// TwinCAT 3 PLC project Untitled1
// ProgramVersion: 3.1.4023.0
// libraries:
//   Tc2_BABasic, * (Beckhoff Automation GmbH)
//   Tc2_ControllerToolbox, * (Beckhoff Automation GmbH)
//   Tc2_MC2, * (Beckhoff Automation GmbH)
//   Tc2_NC, * (Beckhoff Automation GmbH)
//   Tc2_NCI, * (Beckhoff Automation GmbH)
//   Tc2_Standard, * (Beckhoff Automation GmbH)
//   Tc2_System, * (Beckhoff Automation GmbH)
//   Tc2_TempController, * (Beckhoff Automation GmbH)
//   Tc3_Module, * (Beckhoff Automation GmbH)
//   Tc3_mxAutomation, * (Beckhoff Automation GmbH)
//   Tc3_mxAutomationV3_0, * (Beckhoff Automation GmbH)
//   VisuDialogs, * (System)
//   PLC_EposCmdNick,1.0.0.0,TUT
//   VisuSymbols,3.5.10.0,System
// project tree:
//   / GlobalTextList.TcGTLO, PlcTask.TcTTO, Visualization Manager.TcVMO (not stored)
//   GVLs/ GVL_AxisCtrl.TcGVL, GVL_IO.TcGVL, GVL_NC.TcGVL, Scope_Variables.TcGVL
//   POUs/Backup/ PRG_ExtrusionSystem.TcPOU (not stored)
//   POUs/FB/ FB_EnableAxis.TcPOU, FB_EnableNetwork.TcPOU, FB_EPOSstates.TcPOU, FB_EPOS_Control.TcPOU, FB_ExtrusionSystem.TcPOU, FB_SimpleNciSequence.TcPOU, FB_TempControl.TcPOU, FB_ExtrusionSystemRev.TcPOU
//   POUs/ MAIN.TcPOU
//   POUs/Programs/ PRG_AxisControl.TcPOU, PRG_AxesEnable.TcPOU, PRG_ExtruderSys.TcPOU, PRG_ExtruderSys_Alt.TcPOU, PRG_Init.TcPOU, PRG_updateDrives.TcPOU
//   VISUs/ Visualization.TcVIS
// real-time tasks:
//   TASK PlcTask: cycle T#10ms, priority 20, ADS port 350
// motion (NC):
//   TASK NC-Task 1 SAF: cycle T#2ms, priority 4, ADS port 501
//   TASK NC-Task 1 SVB: cycle T#10ms, priority 8, ADS port 511
//   AXIS Axis Th1 (id 1)
//     General: UnitName=°
//     Dynamic: AccelerationMaximum=1500
//     Velo: SlowManual=60, FastManual=80, Maximum=200
//     OtherSettings: AllowMotionCmdToSlave=true, PulseDistancePos=2, PulseDistanceNeg=2
//     encoder EncType=16
//       EncPara: ScaleFactorNumerator=0.000457763671875, MaxCount=#x0000ffff
//         SoftEndMinControl: Enable=true, Range=-16
//         SoftEndMaxControl: Enable=true, Range=35
//     drive DrvType=5
//       Analog: VeloReferenz=220, TorqueSetpointScale=10, ScaleFactorActTorque=0.1
//       TimeComp: TaskDelayCycles=1
//     controller CtrType=1
//       CtrPara: PriorControlFactor=1
//         PosDiffControl: Enable=false
//         PID: PosKp=10
//         Observer: BandWidth=20
//   AXIS Axis Th2 (id 2)
//     General: UnitName=°
//     Velo: SlowManual=60, FastManual=100, Maximum=200
//     OtherSettings: AllowMotionCmdToSlave=true, PulseDistancePos=2, PulseDistanceNeg=2
//     encoder EncType=16
//       EncPara: ScaleFactorNumerator=0.000457763671875, MaxCount=#x0000ffff
//     drive DrvType=5
//       Analog: VeloReferenz=220, TorqueSetpointScale=10, ScaleFactorActTorque=0.1
//       TimeComp: TaskDelayCycles=1
//     controller CtrType=1
//       CtrPara: PriorControlFactor=1
//         PosDiffControl: Enable=false
//         PID: PosKp=10
//         Observer: BandWidth=20
//   AXIS Axis Extruder (id 3)
//     Dynamic: AccelerationMaximum=168, Acceleration=167
//     Velo: RefSearch=10, RefSync=15, SlowManual=10.1, FastManual=15, Maximum=20
//     OtherSettings: AllowMotionCmdToSlave=true
//     encoder EncType=1
//       EncPara: ScaleFactorNumerator=0.000310550364583
//         Inc: RefSoftSyncMask=#x0000ffff
//     drive DrvType=24
//       Analog: VeloReferenz=20, TorqueSetpointScale=10, ScaleFactorActTorque=0.1
//       TimeComp: TaskDelayCycles=1
//     controller CtrType=1
//       CtrPara: PriorControlFactor=1
//         PosDiffControl: Enable=false
//         Observer: BandWidth=20
//   AXIS Axis X (id 4)
//     OtherSettings: AllowMotionCmdToSlave=true
//     encoder EncType=1
//     drive DrvType=5
//       Analog: TorqueSetpointScale=10, ScaleFactorActTorque=0.1
//       TimeComp: TaskDelayCycles=1
//     controller CtrType=1
//       CtrPara: PriorControlFactor=1
//         Observer: BandWidth=20
//   AXIS Axis Z (id 5)
//     OtherSettings: AllowMotionCmdToSlave=true
//     encoder EncType=1
//     drive DrvType=5
//       Analog: TorqueSetpointScale=10, ScaleFactorActTorque=0.1
//       TimeComp: TaskDelayCycles=1
//     controller CtrType=1
//       CtrPara: PriorControlFactor=1
//         Observer: BandWidth=20
//   AXIS Axis Pitch (id 6)
//     OtherSettings: AllowMotionCmdToSlave=true
//     encoder EncType=1
//     drive DrvType=5
//       Analog: TorqueSetpointScale=10, ScaleFactorActTorque=0.1
//       TimeComp: TaskDelayCycles=1
//     controller CtrType=1
//       CtrPara: PriorControlFactor=1
//         Observer: BandWidth=20
//   AXIS Axis Roll (id 7)
//     OtherSettings: AllowMotionCmdToSlave=true
//     encoder EncType=1
//     drive DrvType=5
//       Analog: TorqueSetpointScale=10, ScaleFactorActTorque=0.1
//       TimeComp: TaskDelayCycles=1
//     controller CtrType=1
//       CtrPara: PriorControlFactor=1
//         Observer: BandWidth=20
// I/O:
//   DEVICE Device 2 (EtherCAT), AmsNetId 130.230.11.184.3.1
//     Term 17 (EK1100) [EK1100 EtherCAT Coupler (2A E-Bus)]
//       Term 16 (EL6751) [EL6751 CANopen Master]
//       Term 19 (EL3202) [EL3202 2Ch. Ana. Input PT100 (RTD)]
//       Term 20 (EL1004) [EL1004 4Ch. Dig. Input 24V, 3ms]
//       Term 21 (EL7041) [EL7041 1Ch. Stepper motor output stage (50V, 5A)]
//       Term 22 (EL2004) [EL2004 4Ch. Dig. Output 24V, 0.5A]
//       Term 23 (EL7332) [EL7332 2Ch. DC motor output stage (24V, 1.5A)]
//       Term 22 (EL9011) [EL9011 End Terminal]
//   DEVICE Device 1 (EL6751), AmsNetId 130.230.11.184.2.1
//     Box 2 (EPOS2)
//     Box 3 (EPOS2)
// variable links:
//   NC-Task 1 SAF/Axes/Axis Extruder <-> Device 2 (EtherCAT)/Term 17 (EK1100)/Term 21 (EL7041)
//     Drive/Inputs/In/nState1 @bit 3 <-> STM Status/Status/Error
//     Drive/Inputs/In/nState1 @bit 5 <-> STM Status/Status/Moving negative
//     Drive/Inputs/In/nState1 @bit 4 <-> STM Status/Status/Moving positive
//     Drive/Inputs/In/nState1 @bit 1 <-> STM Status/Status/Ready
//     Drive/Inputs/In/nState1 <-> STM Status/Status/Ready to enable
//     Drive/Inputs/In/nState1 @bit 6 <-> STM Status/Status/Torque reduced
//     Drive/Inputs/In/nState1 @bit 2 <-> STM Status/Status/Warning
//     Drive/Inputs/In/nState2 @bit 3 <-> STM Status/Status/Digital input 1
//     Drive/Inputs/In/nState2 @bit 4 <-> STM Status/Status/Digital input 2
//     Drive/Inputs/In/nState4 @bit 1 <-> WcState/InputToggle
//     Drive/Inputs/In/nState4 <-> WcState/WcState
//     Drive/Outputs/Out/nCtrl1 <-> STM Control/Control/Enable
//     Drive/Outputs/Out/nCtrl1 @bit 2 <-> STM Control/Control/Reduce torque
//     Drive/Outputs/Out/nCtrl1 @bit 1 <-> STM Control/Control/Reset
//     Drive/Outputs/Out/nDataOut2[0] <-> STM Velocity/Velocity
//     Enc/Inputs/In/nDataIn1[0] <-> ENC Status compact/Counter value
//     Enc/Inputs/In/nDataIn2[0] <-> ENC Status compact/Latch value
//     Enc/Inputs/In/nState1 @bit 4 <-> ENC Status compact/Status/Counter overflow
//     Enc/Inputs/In/nState1 @bit 3 <-> ENC Status compact/Status/Counter underflow
//     Enc/Inputs/In/nState1 @bit 7 <-> ENC Status compact/Status/Extrapolation stall
//     Enc/Inputs/In/nState1 <-> ENC Status compact/Status/Latch C valid
//     Enc/Inputs/In/nState1 @bit 1 <-> ENC Status compact/Status/Latch extern valid
//     Enc/Inputs/In/nState1 @bit 2 <-> ENC Status compact/Status/Set counter done
//     Enc/Inputs/In/nState2 @bit 4 <-> ENC Status compact/Status/Status of extern latch
//     Enc/Inputs/In/nState2 <-> ENC Status compact/Status/Status of input A
//     Enc/Inputs/In/nState2 @bit 1 <-> ENC Status compact/Status/Status of input B
//     Enc/Inputs/In/nState2 @bit 2 <-> ENC Status compact/Status/Status of input C
//     Enc/Inputs/In/nState4 @bit 1 <-> WcState/InputToggle
//     Enc/Inputs/In/nState4 <-> WcState/WcState
//     Enc/Outputs/Out/nCtrl1 <-> ENC Control compact/Control/Enable latch C
//     Enc/Outputs/Out/nCtrl1 @bit 3 <-> ENC Control compact/Control/Enable latch extern on negative edge
//     Enc/Outputs/Out/nCtrl1 @bit 1 <-> ENC Control compact/Control/Enable latch extern on positive edge
//     Enc/Outputs/Out/nCtrl1 @bit 2 <-> ENC Control compact/Control/Set counter
//     Enc/Outputs/Out/nDataOut1[0] <-> ENC Control compact/Set counter value
//   NC-Task 1 SAF/Axes/Axis Th1 <-> Device 1 (EL6751)/Box 3 (EPOS2)
//     Enc/Inputs/In/nDataIn1 <-> TxPDO 1/Inputs/PositionActualValue
//   NC-Task 1 SAF/Axes/Axis Th2 <-> Device 1 (EL6751)/Box 2 (EPOS2)
//     Enc/Inputs/In/nDataIn1 <-> TxPDO 3/Inputs/PositionActual
//   Untitled1/Untitled1 Instance <-> Device 1 (EL6751)/Box 2 (EPOS2)
//     PlcTask Inputs/GVL_AxisCtrl.AX1_diStatusWordIs <-> TxPDO 1/Inputs/Status Word
//     PlcTask Inputs/GVL_AxisCtrl.AX2_diVelocityIs <-> TxPDO 4/Inputs/VelocityActual
//     PlcTask Outputs/GVL_AxisCtrl.AX2_diControlWord <-> RxPDO 1/Outputs/ControlWord
//     PlcTask Outputs/GVL_AxisCtrl.Th2_diVeloSet_OUT <-> RxPDO 1/Outputs/TargetVelocity
//   Untitled1/Untitled1 Instance <-> Device 1 (EL6751)/Box 3 (EPOS2)
//     PlcTask Inputs/GVL_AxisCtrl.AX1_diVelocityIs <-> TxPDO 4/Inputs/VelocityActual
//     PlcTask Inputs/GVL_AxisCtrl.AX2_diStatusWordIs <-> TxPDO 1/Inputs/StatusWord
//     PlcTask Outputs/GVL_AxisCtrl.AX1_diControlWord <-> RxPDO 1/Outputs/ControlWord
//     PlcTask Outputs/GVL_AxisCtrl.Th1_diVeloSet_OUT <-> RxPDO 1/Outputs/TargetVelocity
//   Untitled1/Untitled1 Instance <-> Device 2 (EtherCAT)/Term 17 (EK1100)/Term 19 (EL3202)
//     PlcTask Inputs/GVL_IO.lrRawTemp <-> RTD Inputs Channel 1/Value
//   Untitled1/Untitled1 Instance <-> Device 2 (EtherCAT)/Term 17 (EK1100)/Term 20 (EL1004)
//     PlcTask Inputs/GVL_IO.bExcuteButton <-> Channel 1/Input
//   Untitled1/Untitled1 Instance <-> Device 2 (EtherCAT)/Term 17 (EK1100)/Term 22 (EL2004)
//     PlcTask Outputs/GVL_IO.bFan <-> Channel 1/Output
//   Untitled1/Untitled1 Instance <-> Device 2 (EtherCAT)/Term 17 (EK1100)/Term 23 (EL7332)
//     PlcTask Outputs/GVL_IO.bEnableHotend <-> DCM Control Channel 1/Control/Enable
//     PlcTask Outputs/GVL_IO.iHotendPowerLevel <-> DCM Velocity Channel 1/Velocity
//   Untitled1/Untitled1 Instance <-> NC-Task 1 SAF/Axes/Axis Extruder
//     PlcTask Inputs/GVL_NC.Extruder_AXIS.NcToPlc <-> Outputs/ToPlc
//     PlcTask Outputs/GVL_NC.Extruder_AXIS.PlcToNc <-> Inputs/FromPlc
//   Untitled1/Untitled1 Instance <-> NC-Task 1 SAF/Axes/Axis Th1
//     PlcTask Inputs/GVL_AxisCtrl.Th1_iVeloSet_IN <-> Drive/Outputs/Out/nDataOut1[0]
//     PlcTask Inputs/GVL_NC.Th1_AXIS.NcToPlc <-> Outputs/ToPlc
//     PlcTask Outputs/GVL_NC.Th1_AXIS.PlcToNc <-> Inputs/FromPlc
//   Untitled1/Untitled1 Instance <-> NC-Task 1 SAF/Axes/Axis Th2
//     PlcTask Inputs/GVL_AxisCtrl.Th2_iVeloSet_IN <-> Drive/Outputs/Out/nDataOut1[0]
//     PlcTask Inputs/GVL_NC.Th2_AXIS.NcToPlc <-> Outputs/ToPlc
//     PlcTask Outputs/GVL_NC.Th2_AXIS.PlcToNc <-> Inputs/FromPlc
//   Untitled1/Untitled1 Instance <-> NC-Task 1 SAF/Channel 2
//     PlcTask Inputs/MAIN.in_stItpToPlc <-> Outputs/ToPlc
//     PlcTask Outputs/MAIN.out_stPlcToItp <-> Inputs/FromPlc

CONFIGURATION Untitled1
    RESOURCE PLC ON TwinCAT3
        TASK PlcTask(INTERVAL := T#10ms, PRIORITY := 20);
        PROGRAM MAIN WITH PlcTask : MAIN;
        PROGRAM PRG_updateDrives WITH PlcTask : PRG_updateDrives;
    END_RESOURCE
END_CONFIGURATION

// ---- GVLs/GVL_AxisCtrl.TcGVL
{attribute 'qualified_only'}
VAR_GLOBAL
	(********************** Extruder Axis******************************)
	bExtruderSystemEnable 		: BOOL;	
	bExtruderSystemReset 		: BOOL;
	lrHotEndTempSP		 		: LREAL := 200.0;
	sExtruderSystemStatus		: STRING;
	bExtruderReady				: BOOL;
	bExtruderError				: BOOL;

	bExtruder_AxisMoveHMI		: BOOL;
	bExtruder_AxisAbsMoveAct	: BOOL;
	bExtruder_AxisAbsMoveDone	: BOOL;	
	lrExtruder_AxisTarget		: LREAL := 10.0;
	lrExtruder_Retraction		: LREAL := 2.0;
	lrExtruder_AxisVelocity		: LREAL := 2.0;
	
	(******************** Gimbal System *******************************)
	(*Th1 Axis *)
	Th1_iVeloSet_IN AT %I*		:INT;   (*Input Velocity from NC system*)
	Th1_diVeloSet_OUT AT %Q*	:DINT;  (*Velocity Sent to EPOS Drive*)	
	AX1_diVelocityIs AT %I*		:DINT;
	AX1_diPositionIs AT %I*		:DINT;
	AX1_diStatusWordIs AT %I*	:WORD;
	AX1_diControlWord AT %Q*	:WORD;
	
	(*Th2 Axis *)
	Th2_iVeloSet_IN AT %I*		:INT;   (*Input Velocity from NC system*)
	Th2_diVeloSet_OUT AT %Q*	:DINT;  (*Velocity Sent to EPOS Drive*)	
	AX2_diVelocityIs AT %I*		:DINT;
	AX2_diPositionIs AT %I*		:DINT;
	AX2_diStatusWordIs AT %I*	:WORD;
	AX2_diControlWord AT %Q*	:WORD;
	
	(* Combined *)
	bEnableGimbal				: BOOL	:=	FALSE;	(*Running System*)
	bInitDone 					: BOOL	:=	FALSE;	(*Initialisation completed*)
	bAllAxisEnabled				: BOOL	:=	FALSE;	(*Enables axes*)
	bHaltAxes					: BOOL	:=	FALSE;	(*Halt axes*)
	bResetAxes					: BOOL	:=	FALSE; 	(*Reset axes*)
	bZeroAxes					: BOOL	:=	FALSE;
	
	(* Jog *)
	bJogTh1_Pos					: BOOL	:=	FALSE;
	bJogTh1_Neg					: BOOL	:=	FALSE;
	bJogTh2_Pos					: BOOL	:=	FALSE;
	bJogTh2_Neg					: BOOL	:=	FALSE;
	
	(* Move Abs *)
	bExecuteMove 				: BOOL	:=	FALSE;
	lrTh1Target					: LREAL := 0;
	lrTh2Target					: LREAL := 0;
	
END_VAR
VAR_GLOBAL CONSTANT
	NId: STRING:= '130.230.11.184.2.1';		(*ADS ID of CANopen master*)
	Th1_NodeAddr: INT := 3;				(*Node Address of Th1-Axis*)
	Th2_NodeAddr: INT := 2;				(*Node Address of Th1-Axis*)	
END_VAR

// ---- GVLs/GVL_IO.TcGVL
{attribute 'qualified_only'}
VAR_GLOBAL
	lrRawTemp AT %I*			: INT;
	lrHotendTemp 				: LREAL;
	iHotendPowerLevel AT %Q*	: INT;
	bEnableHotend AT %Q*		: BOOL;
	bFan AT %Q*					: BOOL;
	bExcuteButton AT %I*		: BOOL;
END_VAR

// ---- GVLs/GVL_NC.TcGVL
{attribute 'qualified_only'}
VAR_GLOBAL
	(************************* Axis Ref *******************************)
	(* Extruder System *)
	Extruder_AXIS			: AXIS_REF;
	HotEnd_AXIS				: AXIS_REF;	
	(* Gimbal *)
	Th1_AXIS				: AXIS_REF;
	Th2_AXIS				: AXIS_REF;
	
	(************************* Axis Status ****************************)
	(* Extruder System *)
	Extruder_AXIS_Status	: ST_AxisStatus;
	HotEnd_AXIS_Status		: ST_AxisStatus;
	(* Gimbal *)
	Th1_AXIS_Status			: ST_AxisStatus;
	Th2_AXIS_Status			: ST_AxisStatus;
		
	// 	From Niko Code
	//	PlcToNc_Th1 AT %Q*		: PLCTONC_AXIS_REF;	(*Motor 1*)
	//	NcToPlc_Th1 AT %I*		: NCTOPLC_AXIS_REF;	(*Motor 1*)
	
END_VAR

// ---- GVLs/Scope_Variables.TcGVL
{attribute 'qualified_only'}
VAR_GLOBAL
	fX_Scope	: LREAL;
	fY_Scope	: LREAL;
	fW_Scope	: LREAL;
END_VAR

// ---- POUs/MAIN.TcPOU
PROGRAM MAIN
VAR
	Hearbeat				: DINT :=0;
	lrHotendTemp			: LREAL;
	bEnableExtrusionSystem 	: BOOL := FALSE;
	bResetExtrusionSystem 	: BOOL := FALSE;
	bEnableGimbalAxis 		: BOOL := FALSE;
	
	fUserOverride			: LREAL:= 100.0;
	in_stItpToPlc	AT %I*:	NcToPlc_NciChannel_Ref;
	out_stPlcToItp	AT %Q*:	PLCTONC_NCICHANNEL_REF;
	
	fbSimpleNciSequence		: FB_SimpleNciSequence;
	bExecSimpleNci:	BOOL	:= FALSE;
	
END_VAR

Hearbeat := Hearbeat+1;
bExecSimpleNci := GVL_IO.bExcuteButton;
GVL_IO.lrHotendTemp := GVL_IO.lrRawTemp/10.0;

//PRG_ExtruderSys();
PRG_ExtruderSys_Alt();

//IF NOT  PRG_Init.BDONE THEN
IF NOT GVL_AxisCtrl.bInitDone THEN
	PRG_Init(bExecute:=TRUE , bDone=>GVL_AxisCtrl.bInitDone);
	//GVL_AxisCtrl.bEnableAxes := FALSE;
ELSE	(*Init done*)

PRG_AxesEnable(
	bEnable:= GVL_AxisCtrl.bEnableGimbal,
	bHalt:= GVL_AxisCtrl.bHaltAxes,
	bReset:= GVL_AxisCtrl.bResetAxes,
	bAxesEnabled=> GVL_AxisCtrl.bAllAxisEnabled, 
	bFaultActive=> , 
	wEnabledStates=> , 
	wFaultStates=> );
	
PRG_AxisControl();
		
ItpSetOverridePercent(fOverridePercent:=fUserOverride , sPlcToNci:=out_stPlcToItp);

fbSimpleNciSequence(
	bExecute:= bExecSimpleNci, 
	bBusy=> , 
	bError=> , 
	bDone=> , 
	stX:=GVL_NC.Th1_AXIS, 
	stY:=GVL_NC.Th2_AXIS, 
	stZ:=GVL_NC.Th2_AXIS, 
	stItpToPlc:= in_stItpToPlc , 
	stPlcToItp:= out_stPlcToItp);		
END_IF;	
	
	
//PRG_ExtrusionSystem(
//	bEnable:= bEnableExtrusionSystem,
//	bReset := bResetExtrusionSystem);

END_PROGRAM

// ---- POUs/FB/FB_SimpleNciSequence.TcPOU
FUNCTION_BLOCK FB_SimpleNciSequence
VAR_INPUT
	bExecute			: BOOL;
END_VAR
VAR_OUTPUT
	bBusy				: BOOL;
	bError				: BOOL;
	bDone				: BOOL;
END_VAR
VAR_IN_OUT
	stX					: AXIS_REF;
	stY					: AXIS_REF;
	stZ					: AXIS_REF;
	stItpToPlc			: NCTOPLC_NCICHANNEL_REF;
	stPlcToItp			: PLCTONC_NCICHANNEL_REF;
END_VAR
VAR
	nState				: UDINT	:= 0;
	nErrorState			: UDINT;
	
	fbBuildGroup		: CfgBuild3DGroup;
	fbLoadGCode			: ItpLoadProgEx;
	fbStartGCode		: ItpStartStopEx;
	fbClearGroup		: CfgReconfigGroup;
	fbConfirmHsk		: ItpConfirmHsk;
	
	nInterpreterState	: UDINT	:= 0;
	bConfirmHsk			: BOOL	:= FALSE;
	
	sPrgName			: STRING(255) := 'C:\Temp\github\RPW_PMJ_Group\PMJ_Cellv2\first.nc';
END_VAR

CASE nState OF
0:
	IF bExecute THEN
		bBusy	:= TRUE;
		bDone	:= FALSE;
		bError	:= FALSE;
		nErrorState	:= nState;
		nState	:= 10;
	END_IF	
	
10:
	// first build interpolation group 
	fbBuildGroup(
		bExecute:=TRUE, 
		nGroupId:=ItpGetGroupId(sNciToPlc:=stItpToPlc) , 
		nXAxisId:=stX.NcToPlc.AxisId, 
		nYAxisId:=stY.NcToPlc.AxisId, 
		nZAxisId:=0,
//		nZAxisId:=stZ.NcToPlc.AxisId, 
//		nQ1AxisId:= 0, 
//		nQ2AxisId:= 0, 
//		nQ3AxisId:= 0, 
//		nQ4AxisId:= 0, 
//		nQ5AxisId:= 0, 
		tTimeOut:= , 
		bBusy=> , 
		bErr=> , 
		nErrId=> );
	IF NOT fbBuildGroup.bBusy THEN
		IF NOT fbBuildGroup.bErr THEN
			nState	:= 20;
		ELSE
			(* add error handling *)
			nErrorState	:= nState;
			bBusy	:= FALSE;
			bError	:= TRUE;
			nState	:= 9999;
		END_IF
		fbBuildGroup(bExecute:=FALSE); 
	END_IF
	
20:
	// load g-code file 
	// pls. ensure that first.nc is available in TwinCAT\MC\NCI-folder 
	fbLoadGCode(
		sNciToPlc:=stItpToPlc, 
		bExecute:=TRUE, 
		sPrg:= sPrgName, 
		nLength:= INT_TO_UDINT(LEN(sPrgName)), 
		tTimeOut:= , 
		bBusy=> , 
		bErr=> , 
		nErrId=> );
	IF NOT fbLoadGCode.bBusy THEN
		IF NOT fbLoadGCode.bErr THEN
			nState	:= 30;
		ELSE
			(* add error handling *)
			nErrorState	:= nState;
			bBusy	:= FALSE;
			bError	:= TRUE;
			nState	:= 9999;				
		END_IF
		fbLoadGCode(sNciToPlc:=stItpToPlc, bExecute:=FALSE); 
	END_IF
	
30:
	// we have to check the status of the interpreter. It has to be in ready state, in case of loading the program successfully.
	nInterpreterState	:= ItpGetStateInterpreter(sNciToPlc:=stItpToPlc);
	IF nInterpreterState = Tc2_NCI.NCI_INTERPRETER_READY THEN
		nState	:= 40;
	ELSE
		(* add error handling *)
		nErrorState	:= nState;
		bBusy	:= FALSE;
		bError	:= TRUE;
		nState	:= 9999;				
	END_IF
	
40:
	// start g-code file
	fbStartGCode(
		bStart:=TRUE, 
		bStop:=FALSE, 
		tTimeOut:= , 
		sNciToPlc:= stItpToPlc, 
		bBusy=> , 
		bErr=> , 
		nErrId=> );
	IF NOT fbStartGCode.bBusy THEN
		IF NOT fbStartGCode.bErr THEN
			nState	:= 50;
		ELSE	
			(* add error handling *)
			nErrorState	:= nState;
			bBusy	:= FALSE;
			bError	:= TRUE;
			nState	:= 9999;				
		END_IF
		fbStartGCode( bStart:=FALSE, sNciToPlc:= stItpToPlc ); 
	END_IF
	
50:
	// check state, again - we are at least not in ready state for several ticks
	// this is to ensure that we don't indicate program has finished, before we have started 
	nInterpreterState	:= ItpGetStateInterpreter(sNciToPlc:=stItpToPlc);
	IF nInterpreterState <> Tc2_NCI.NCI_INTERPRETER_READY THEN
		// nci is running
		nState	:= 60;
	END_IF

60:
	nInterpreterState	:= ItpGetStateInterpreter(sNciToPlc:=stItpToPlc);
	IF	nInterpreterState = Tc2_NCI.NCI_INTERPRETER_READY THEN
		// program has finished
		nState	:= 70;
	ELSIF nInterpreterState = Tc2_NCI.NCI_INTERPRETER_ABORTED THEN
		// a run-time error occured - this could be a lag error or something else... 
		// add error handling
		;
	END_IF	
70:
	// program has finished 
	// now clear interpolation group 
	fbClearGroup(
		bExecute:=TRUE, 
		nGroupId:=ItpGetGroupId(sNciToPlc:=stItpToPlc) , 
		tTimeOut:= , 
		bBusy=> , 
		bErr=> , 
		nErrId=> );
	IF NOT fbClearGroup.bBusy THEN
		IF NOT fbClearGroup.bErr THEN
			nState	:= 80;
		ELSE
			(* add error handling *)
			nErrorState	:= nState;
			bBusy	:= FALSE;
			bError	:= TRUE;
			nState	:= 9999;				
		END_IF
		fbClearGroup(bExecute:=FALSE); 
	END_IF
80:
	bDone	:= TRUE;
	bBusy	:= FALSE;
	IF NOT bExecute THEN
		nState	:= 0;
	END_IF
9999:
	// error state 
	IF NOT bExecute THEN
		nState	:= 0;
		bError	:= FALSE;
	END_IF
END_CASE

// handling of m-functions is done outside statemachine
// all m-functions are directly confiremd. In a real application we have of course to consider the m-function numbers to turn on/off certain functions in the machine.
IF ItpIsHskMFunc(stItpToPlc) AND NOT fbConfirmHsk.bBusy THEN
	bConfirmHsk	:= TRUE;
ELSE	
	bConfirmHsk	:= FALSE;
END_IF	

fbConfirmHsk(
	bExecute:=bConfirmHsk , 
	sNciToPlc:=stItpToPlc , 
	sPlcToNci:=stPlcToItp , 
	bBusy=> , 
	bErr=> , 
	nErrId=> );

END_FUNCTION_BLOCK

// ---- POUs/Programs/PRG_ExtruderSys_Alt.TcPOU
PROGRAM PRG_ExtruderSys_Alt
VAR
	fbExtrusionSystem: FB_ExtrusionSystemRev;
END_VAR

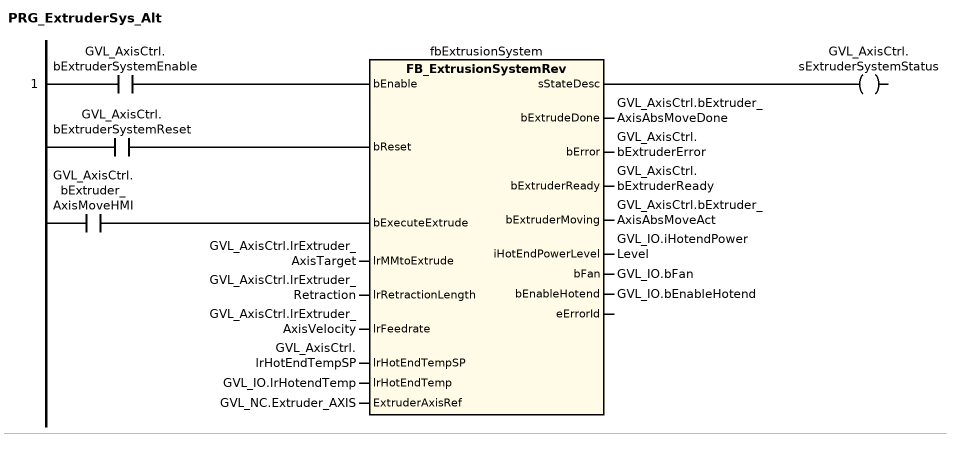
// NETWORK 1
fbExtrusionSystem(
    bEnable := GVL_AxisCtrl.bExtruderSystemEnable,
    bReset := GVL_AxisCtrl.bExtruderSystemReset,
    bExecuteExtrude := GVL_AxisCtrl.bExtruder_AxisMoveHMI,
    lrMMtoExtrude := GVL_AxisCtrl.lrExtruder_AxisTarget,
    lrRetractionLength := GVL_AxisCtrl.lrExtruder_Retraction,
    lrFeedrate := GVL_AxisCtrl.lrExtruder_AxisVelocity,
    lrHotEndTempSP := GVL_AxisCtrl.lrHotEndTempSP,
    lrHotEndTemp := GVL_IO.lrHotendTemp,
    ExtruderAxisRef := GVL_NC.Extruder_AXIS,
    bExtrudeDone => GVL_AxisCtrl.bExtruder_AxisAbsMoveDone,
    bError => GVL_AxisCtrl.bExtruderError,
    bExtruderReady => GVL_AxisCtrl.bExtruderReady,
    bExtruderMoving => GVL_AxisCtrl.bExtruder_AxisAbsMoveAct,
    iHotEndPowerLevel => GVL_IO.iHotendPowerLevel,
    bFan => GVL_IO.bFan,
    bEnableHotend => GVL_IO.bEnableHotend); // FB_ExtrusionSystemRev
GVL_AxisCtrl.sExtruderSystemStatus := fbExtrusionSystem.sStateDesc;

END_PROGRAM

// ---- POUs/FB/FB_ExtrusionSystemRev.TcPOU
FUNCTION_BLOCK FB_ExtrusionSystemRev
VAR_INPUT
	bEnable 			: BOOL;
	bReset 				: BOOL;
	bExecuteExtrude		: BOOL;
	lrMMtoExtrude  		: LREAL;
	lrRetractionLength	: LREAL;
	lrFeedrate   		: LREAL;
	lrHotEndTempSP		: LREAL;
	lrHotEndTemp 		: LREAL;	
END_VAR
VAR_OUTPUT
	sStateDesc			: STRING;
	bExtrudeDone 	    : BOOL;
	bError				: BOOL;
	bExtruderReady		: BOOL;
	bExtruderMoving		: BOOL;
	iHotEndPowerLevel 	: INT;
	bFan				: BOOL;
	bEnableHotend		: BOOL;
	eErrorId			: UDINT;
END_VAR
VAR_IN_OUT
	ExtruderAxisRef			: AXIS_REF;
END_VAR
VAR
	nState					: UDINT := 0;
	nErrorState				: UDINT;
		
	RTrig_Reset				: R_TRIG;
	MC_Power_Extruder		: MC_Power;
	MC_Reset_Extruder 		: MC_Reset;
	MC_ZeroPos_Extruder		: MC_SetPosition;
	MC_Stop_Extruder 		: MC_Stop;
	MC_Move_Rel_Extruder 	: MC_MoveRelative;
	fbHotendTempController 	: FB_TempControl;
	
	bHeating				: BOOL := FALSE;
	bAtTempSP				: BOOL := FALSE;
	bMoveRelative			: BOOL := FALSE;
	fbSetPos				: MC_SetPosition;
	lrExtrudeDist  			: LREAL;
END_VAR

ExtruderAxisRef.ReadStatus();
RTrig_Reset(CLK:=bReset , Q=> );

MC_Power_Extruder(
	Axis:= ExtruderAxisRef, 
	Enable:= bExtruderReady, 
	Enable_Positive:= bExtruderReady, 
	Enable_Negative:= bExtruderReady, 
	Override:= , 
	BufferMode:= , 
	Options:= , 
	Status=> , 
	Busy=> , 
	Active=> , 
	Error=> bError, 
	ErrorID=> eErrorId);
	
fbHotendTempController(
		bEnableHeater:= bEnableHotEnd, 
		lrPV:= lrHotendTemp, 
		lrSP:= lrHotEndTempSP, 
		iOutput=> iHotEndPowerLevel, 
		bError=>bError, 
		eErrorId=> eErrorId,
		bEnableHotend=> bEnableHotend);
		
MC_Move_Rel_Extruder(
	Axis:= ExtruderAxisRef, 
	Execute:= bMoveRelative, 
	Distance:= lrExtrudeDist, 
	Velocity:= lrFeedrate, 
	Acceleration:= , 
	Deceleration:= , 
	Jerk:= , 
	BufferMode:= , 
	Options:= , 
	Done=> bExtrudeDone, 
	Busy=> , 
	Active=> bExtruderMoving , 
	CommandAborted=> , 
	Error=> bError, 
	ErrorID=> eErrorId);
	
//IF NOT bEnable THEN
//	nState := 10;
//END_IF

IF RTrig_Reset.CLK THEN
	nState := 100;
END_IF

IF lrHotendTemp >= (lrHotEndTempSP*0.98) THEN
	bAtTempSP := TRUE;
ELSE
	bAtTempSP := FALSE;
END_IF

	
CASE nState OF
	0:	// init
		sStateDesc := 'FB INIT';
		bExtrudeDone := FALSE;
		bError := FALSE;
		bExtruderMoving := FALSE;
		//GVL_AxisCtrl.bExtruder_AxisAbsMove := FALSE;
		iHotEndPowerLevel := 0;
		bFan := FALSE;
		nState := 10;
		
	10: // idle
		sStateDesc := 'IDLE';
		iHotEndPowerLevel := 0;
		bEnableHotEnd := FALSE;
		bExtruderReady := FALSE;
		bFan := FALSE;
		IF bEnable THEN 
			nState := 20;
		END_IF		

	20: // Turn on heater
		IF NOT bEnable THEN
			nState := 10;
		END_IF
		
		sStateDesc := 'START HEATING';
		bFan := TRUE;			
		bEnableHotend := TRUE;
		nState := 30;
		
	30: // Heating
		IF NOT bEnable THEN
			nState := 10;
		END_IF
		sStateDesc := 'HEATING TO REACH OPERATING TEMP';
		IF bAtTempSP THEN
			nState := 40;
		ELSE
			bExtruderReady := FALSE;	
		END_IF
		
	40: // Ready to Extrude
		IF NOT bEnable THEN
			nState := 10;
		END_IF
		
		IF bAtTempSP THEN
			sStateDesc := 'WAITING FOR MOVE COMMAND';
			bExtruderReady := TRUE;
			IF bExecuteExtrude THEN;
				nState := 50;
			END_IF
		ELSE
			bExtruderReady := FALSE;
			nState := 30;
		END_IF
		
	50: // Move Relative
		IF NOT bEnable THEN
			nState := 10;
		END_IF
		sStateDesc := 'EXTRUDING';
		lrExtrudeDist := lrMMtoExtrude;
		bMoveRelative := TRUE;
		IF bExtrudeDone THEN (* Requested Distance Extruded *)
			bExtrudeDone 	:= FALSE;
			bMoveRelative 	:= FALSE;
			nState := 60;
		END_IF
	60: // Retract
		sStateDesc := 'RETRACTING';
		IF NOT bEnable THEN
			nState := 10;
		END_IF
		lrExtrudeDist := lrRetractionLength * -1; (* Retract *)
		bMoveRelative := TRUE;
		IF bExtrudeDone THEN (* Requested Retraction Done *)
			bExtrudeDone 	:= FALSE;
			bMoveRelative 	:= FALSE;
			nState := 40;
		END_IF
			
	100: // Reset
		sStateDesc := 'RESET EXTRUDER AXIS';
		MC_Reset_Extruder(Axis:=ExtruderAxisRef, Execute:=TRUE);
		IF MC_Reset_Extruder.Done THEN
			nState := 10;
		END_IF
	999: //Error	
		
	ELSE
	sStateDesc := 'INVALID STATE';
	nState := 0;
END_CASE

END_FUNCTION_BLOCK

// ---- POUs/FB/FB_TempControl.TcPOU
FUNCTION_BLOCK FB_TempControl
VAR_INPUT
	bEnableHeater 		: BOOL;
	lrPV 			: LREAL;    (*Process Variable *)
	lrSP 			: LREAL;	(*Set Point *)
END_VAR
VAR_OUTPUT
	bEnableHotend	: BOOL := FALSE;		(* Enable EL7332-DCM Control Ch1*)
	iOutput 		: INT;		(* Output-INT set to EL7332 DCM Velocity Ch1*)
	bError 			: BOOL;
	eErrorId 		: E_CTRL_ErrorCodes;
END_VAR
VAR
	eCTRL_Mode 				: E_CTRL_MODE := eCTRL_MODE_Tune; 	(*   eCTRL_MODE_TUNE  ;*)
	bSelSetpoint			: BOOL:= FALSE;
	fW1						: LREAL;				(* first setpoint *)
	fW2						: LREAL;				(* second setpoint - standby setpoint*)
	fY						: LREAL;						(* control value *)
	fX						: LREAL;						(* actual value from simulated process *)
	bYPWMPos				: BOOL;
	bYPWMNeg				: BOOL;

	(************************** Controller Parameters structure ****************************************)
	stControllerParameter	: ST_CTRL_TempCtrlParameter := (		
		(* general parameters *)
		iMode					:= 1,											(* 1=heating, 2=cooling, 3=heating&cooling *)
		iReactionOnFailure		:= eCTRL_ReactionOnFailure_StopController,		(* 0=controller off, 1=manual op, 2=yMin, 3=yMax *)
	
		bSelCtrlParameterSet	:= FALSE,			(* FALSE = internal set, TRUE = external set *)
	
		dwAlarmSupp				:= 16#0000EFFF,		(* alarm suppression *)
		tCtrlCycleTime			:= T#500MS,			(* controller cycle time *)
		tTaskCycleTime			:= T#10MS,			(* plc task cycle time *)
		
		(* tuning parameters *)
		iTuningMode				:= 1,				(* only heating, only cooling, first heating then cooling or vice versa *)
	
		tTuneStabilisation		:= T#1S,			(* wait for a stable system *)
		fEndTunePercentHeating	:= 80.0,			(* switch to closed loop control when X > 0.8*W *)
		fYTuneHeating			:= 31000,			(* step change while tuning operation *)
		fYStableHeating			:= 0.0,				(* tuning operation *)
	
		fEndTunePercentCooling	:= 20.0,			(* switch to closed loop control when X < 0.2*W *)
		fYTuneCooling			:= 0.0,				(* step change while tuning operation *)
		fYStableCooling			:= 0.0,				(* tuning operation *)
		fScalingFactor			:= 1.0,				(* Scaling factor for KP heating/cooling *)
		
		(* setpoint parameters *)
		fWMin					:= 0.0,				(* lower limit *)
		fWMax					:= 250.0,			(* upper limit *)
	
		(* start up *)
		bEnableSoftStart		:= FALSE,			(* FALSE = no soft start, TRUE = soft start *)
		bEnableRamping			:= FALSE,		    (* FALSE = no ramping, TRUE = ramping *)
	
		fWStartUp				:= 0.0,				(* soft start plateau setpoint *)
		tStartUp				:= T#0MS,			(* soft start waiting time*)
		bStartUpRamping			:= FALSE,			(* enable ramping while start up phase *)
		fWStartUpVeloPos		:= 1.0,				(* max gradient for increasing setpoint in start up phase*)
		fWStartUpVeloNeg		:= 1.0,				(* max gradient for decreasing setpoint in start up phase *)
	
		fWVeloPos				:= 1.0,				(* max gradient for increasing setpoint *)
		fWVeloNeg				:= 1.0,				(* max gradient for decreasing setpoint *)	
	
		(* actual value parameters *)
		bFilter 				:= FALSE,
		tFilter					:= T#0S,
		
		(* deadband parameters *)
		bDeadband				:= FALSE,
		fEDeadband				:= 0.0,				(* deadband *)
		
		(* control value parameters*)
		fYMin					:= 0,				(* lower limit *)
		fYMax					:= 32000,			(* upper limit *)
		fYManual				:= 0.0,				(* manual operation*)
		fYOnFailure				:= 0.0,				(* control value on failure *)
		
		tPWMCycleTime			:= T#1S,										(* PWM: period *)
		tPWMMinOffTime			:= t#0s,										(* PWM: min off time *)
		tPWMMinOnTime			:= t#0s,										(* PWM: min on time *)
		tPWMWaitingTime			:= t#0s,										(* PWM: min waiting time *) (* not yet implemented !!!!*)
		
		fYThresholdOff			:= 0.0,				(* 3-Point: Off threshold *)
		fYThresholdOn			:= 0.0,				(* 3-Point: On threshold *)
	
		nCyclesForSwitchOver	:= 100,
	
		(* controller settings *)
		bEnablePreController 	:= FALSE,			(* enable precontroller *)
		bEnableZones 			:= FALSE,			(* enable zone around setpoint with open loop control *)
		bEnableCVFilter 		:= FALSE,			(* enable filter for CV (type see iFilterType) *)
		iFilterType 			:= E_FilterType_FIRSTORDER,		(* filtertype of CV filter *)
		iControllerType 		:= eCTRL_ControllerType_PID,	(* used controller normally PID *)
		
		
		(* min max temperatures	*)
		
		TempLowLow				:= 5.0,
		TempLow					:= 10.0,
		TempHigh				:= 205.0,
		TempHighHigh			:= 225.0,
		TempAbsoluteHigh		:= 240.0,
		TempAbsoluteLow			:= 5.0,	
		
		(* internal tuning parameters *)
		fTuneKp					:= 1.0,
		fTuneTn					:= 2.5,
		fTuneTv					:= 0.42,
		fTuneTd					:= 0.25
		);
	
	(* Other Function Blocks *)
	fbTempController			: FB_CTRL_TempController;	
	fbCtrlParameter				: FB_CTRL_CtrlParameter;
	stController				: ST_CTRL_ParaController;
	
	(* Debug *)
	fMaxOvershoot			: LREAL;
	tStartUpTime			: TIME;
	eCtrlState				: E_CTRL_STATE;
	
END_VAR


// Heater is Enabled
IF bEnableHeater THEN  
	(* Start controller *)
	fbTempController(
						eCtrlMode				:= eCTRL_Mode, 
						bSelSetpoint			:= bSelSetpoint, 
						fW1						:= lrSP, 
						fW2						:= lrSP-30, 
						fX						:= lrPV, 
						fYManual				:= , 
						bOpenThermocouple		:= FALSE, 
						bReverseThermocouple	:= FALSE, 
						bBackVoltage			:= FALSE, 
						bLeakage				:= FALSE, 
						bShortCircuit			:= FALSE, 
						bOpenCircuit			:= FALSE, 
						sParaControllerExternal	:= stController, 
						sControllerParameter	:= stControllerParameter, 
						);
						
	(* Analog output *)			
	fY := fbTempController.fYAnalog;
	
	bError := fbTempController.bError;
	eErrorId := fbTempController.eErrorId;
	
	(* Choose set of controller parameters *)
	IF fbTempController.eCtrlState = eCTRL_STATE_TUNED THEN
		eCTRL_Mode := eCTRL_MODE_ACTIVE;	
	END_IF
	
	(* Debug *)
	fMaxOvershoot := fbTempController.fMaxOverShoot;
	tStartUpTime := fbTempController.tStartUpTime;
	
	(* Scope *)
	Scope_Variables.fW_Scope:= lrSP;
	Scope_Variables.fX_Scope := fX;
	Scope_Variables.fY_Scope := fY;
	
	(*FB Outputs *)
	bEnableHotend := TRUE;
	iOutput := REAL_TO_INT(fY);

ELSE // Heater Disabled
	bEnableHotend := FALSE;
	iOutput := 0;
	fbTempController(
		eCtrlMode				:= eCTRL_MODE_IDLE, 
		fW1						:= 0,
		sControllerParameter	:= stControllerParameter,
		);
END_IF

END_FUNCTION_BLOCK

// ---- POUs/Programs/PRG_Init.TcPOU
PROGRAM PRG_Init
VAR_INPUT
	bExecute				: BOOL;		(*Executes initialisation*)
END_VAR
VAR_OUTPUT
	bDone					: BOOL;		(*Initialisation Completed*)
END_VAR
VAR
	fbEnableNetwork_Th1		: FB_EnableNetwork;
	fbEnableNetwork_Th2		: FB_EnableNetwork;
	fbSetVelocityProfile_Th1: FB_SetVelocityProfile;
	fbSetVelocityProfile_Th2: FB_SetVelocityProfile;

	R_DoneTrigger_Th1		: R_TRIG;	(*Bus and controllers has been enabled*)
	R_DoneTrigger_Th2		: R_TRIG;
	
	bSetVeloProfDone		: BOOL	:= FALSE;
	bBusEnabled				: BOOL	:= FALSE;(*Bus and controllers are enabled*)
END_VAR

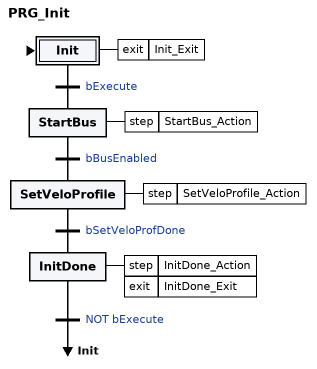
INITIAL_STEP Init:
    Init_Exit(P0);  // exit action
END_STEP
TRANSITION FROM Init TO StartBus
    := bExecute;
END_TRANSITION
STEP StartBus:
    StartBus_Action(N);  // step action
END_STEP
TRANSITION FROM StartBus TO SetVeloProfile
    := bBusEnabled;
END_TRANSITION
STEP SetVeloProfile:
    SetVeloProfile_Action(N);  // step action
END_STEP
TRANSITION FROM SetVeloProfile TO InitDone
    := bSetVeloProfDone;
END_TRANSITION
STEP InitDone:
    InitDone_Action(N);  // step action
    InitDone_Exit(P0);  // exit action
END_STEP
TRANSITION FROM InitDone TO Init
    := NOT bExecute;
END_TRANSITION

ACTION Init_Exit:
bDone := FALSE;
END_ACTION

ACTION InitDone_Action:
bDone :=TRUE;
END_ACTION

ACTION InitDone_Exit:
bDone :=FALSE;
END_ACTION

ACTION SetVeloProfile:

END_ACTION

ACTION SetVeloProfile_Action:
fbSetVelocityProfile_Th1(
	ADSNetId:= GVL_AxisCtrl.NId ,
	NodeId:=  GVL_AxisCtrl.Th1_NodeAddr,
	Write:= TRUE,
	ProfileAcceleration:= 100000,
	ProfileDeceleration:= 100000,
	Done=> , 
	Err=> , 
	ErrNo=> );
	
fbSetVelocityProfile_Th2(
	ADSNetId:= GVL_AxisCtrl.NId ,
	NodeId:=  GVL_AxisCtrl.Th2_NodeAddr,
	Write:= TRUE,
	ProfileAcceleration:= 100000,
	ProfileDeceleration:= 100000,
	Done=> , 
	Err=> , 
	ErrNo=> );
	
//R_DoneTrigger_Th1(CLK:=fbSetVelocityProfile_Th1.Done , Q=> );
//R_DoneTrigger_Th2(CLK:=fbSetVelocityProfile_Th2.Done , Q=> );

//IF R_DoneTrigger_Th1.Q AND R_DoneTrigger_Th2. THEN
IF fbSetVelocityProfile_Th1.Done AND fbSetVelocityProfile_Th1.Done THEN
	bSetVeloProfDone := TRUE;
ELSE
	bSetVeloProfDone := FALSE;
END_IF;
END_ACTION

ACTION StartBus_Action:
(*Anabloidaan akselit. Mode: 16#03	= 	ProfileVelocityMode*)
fbEnableNetwork_Th1(
	ADSNetId:= GVL_AxisCtrl.NId,
	NodeId:= GVL_AxisCtrl.Th1_NodeAddr,
	bExcute:= TRUE,
	bEnabled:= TRUE,
	iOpMode:= 16#03,
	bDone=> , 
	bErr=> ,
	iErrNo=> );
	
fbEnableNetwork_Th2(
	ADSNetId:= GVL_AxisCtrl.NId,
	NodeId:= GVL_AxisCtrl.Th2_NodeAddr,
	bExcute:= TRUE,
	bEnabled:= TRUE,
	iOpMode:= 16#03,
	bDone=> , 
	bErr=> ,
	iErrNo=> );
	

R_DoneTrigger_Th1(CLK:=fbEnableNetwork_Th1.bDone , Q=> );
R_DoneTrigger_Th2(CLK:=fbEnableNetwork_Th2.bDone , Q=> );

IF R_DoneTrigger_Th1.Q AND R_DoneTrigger_Th2.Q THEN
	bBusEnabled := TRUE;
ELSE
	bBusEnabled := FALSE;
END_IF;

(*Initialisation completed*)
//GVL_AxisCtrl.bInitDone := fbEnableNetwork.bDone;
END_ACTION

END_PROGRAM

// ---- POUs/FB/FB_EnableNetwork.TcPOU
FUNCTION_BLOCK FB_EnableNetwork
VAR_INPUT
	ADSNetId		: STRING; 	(* Adress of the CANOpen Master. *)
	NodeId			: INT;		(* Represents the node adress witch is found on Dip Switch of Device *)
	bExcute			: BOOL;		(* Excutes and updates the operation*)
	bEnabled		: BOOL;		(* Is axis enabled?*)
	iOpMode			: INT;		(*Operation Mode. See PLC_EposCmd.lib:FB_SetOperationMode for modes
										16#01	= 	ProfilePositonMode
										16#03	= 	ProfileVelocityMode
										16#06	= 	HomingMode
										16#FF	= 	PositonMode
										16#FE	= 	VelocityMode
										16#FD	= 	CurrentMode*)
END_VAR
VAR_OUTPUT
	bDone			: BOOL;		(* Done Flag is set when Function has done*)
	bErr			: BOOL;		(* Err Flag is TRUE if an Error has accured, see iErrno for more Details *)
	iErrNo			: UDINT;		(* Contains detailed Error Information*)
END_VAR
VAR
	iStep: UINT 	:= 0;		(*stepper*)
	fbClearFault	: FB_ClearFault;
	fbSetOPMode		: FB_SetOperationMode;
	fbEnable		: FB_SetEnableState;
	fbDisable		: FB_SetDisableState;
END_VAR

CASE iStep OF
1:	(* Init *)
	bExcute := FALSE;
	bDone := FALSE;
	bErr := FALSE;
	iErrNo := 0;
	iStep := 100;

100:	(*Activate node*)
	fbClearFault(
		ADSNetId:=ADSNetId ,
		NodeId:= NodeId,
		Write:= TRUE,
		Done=> ,
		Err=> ,
		ErrNo=> );
	fbSetOPMode(
		ADSNetId:=ADSNetId ,
		NodeId:= NodeId,
		Write:= fbClearFault.Done,
		Mode:= INT_TO_SINT(iOpMode),
		Done=> ,
		Err=>bErr,
		ErrNo=>iErrNo);
		
	IF fbSetOPMode.Err THEN
		iStep := 0;
	ELSE
		IF fbSetOPMode.Done THEN
			iStep:=200;
		END_IF;
	END_IF;

200: (*Enable or Disable Node*)
	IF bEnabled THEN
		fbEnable(
			ADSNetId:=ADSNetId ,
			NodeId:= NodeId,
			Write:= TRUE,
			Done=> ,
			Err=> bErr,
			ErrNo=> iErrNo);
	ELSE
		fbDisable(
			ADSNetId:=ADSNetId ,
			NodeId:= NodeId,
			Write:= TRUE,
			Done=> ,
			Err=> bErr,
			ErrNo=> iErrNo);
	END_IF;

	IF bErr THEN
		iStep:=0;
	ELSE
		IF (fbEnable.Done OR fbDisable.Done) THEN
			iStep:=9999;
		END_IF;
	END_IF;

9999: (*DONE*)
	bDone := TRUE;
	iStep := 0;

ELSE
	IF bExcute THEN
		iStep := 1;
		bDone := FALSE;
	END_IF;

END_CASE;

(*
*********************WRITE******************************************
	Done			: BOOL;		(* Done Flag is set when Function has done *)
	Err				: BOOL;		(* Err Flag is TRUE if an Error has accured, see Errno for more Details *)
	ErrNo			: UDINT;		(* Contains detailed Error Information *)
CASE iStep OF

1:	(* Init *)
	Write := FALSE;
	Done := FALSE;
	Err := FALSE;
	ErrNo := 0;
	WriteObj(WRITE := FALSE);
	iStep := 100;

100:	(* Write Mode *)
	WriteObj(
		NETID := ADSNetId,
		PORT := 16#1000 + NodeId,
		IDXGRP := 16#6060,
		IDXOFFS := 0,
		LEN := 1,
		SRCADDR := ADR(Mode),
		WRITE := TRUE,
		TMOUT := t#100ms);
	iStep := 101;
101: WriteObj;
	IF NOT WriteObj.Busy THEN
		iStep := 102 ;
	END_IF
102:	IF WriteObj.Err THEN
		iStep := 0;
		ErrNo := WriteObj.ErrId;
		Multiplexor := 16#606000;
		Err := TRUE;
	ELSE
		iStep := 0;
	END_IF
	Done := TRUE;

ELSE
	IF Write THEN
		iStep := 1;
		Done := FALSE;
	END_IF;
END_CASE;


****************************READ*******************************
CASE iStep OF

1:	(* Init *)
	Read := FALSE;
	Done := FALSE;
	Err := FALSE;
	ErrNo := 0;
	ReadObj(READ := FALSE);
	iStep := 100;

100:	(* Read Object *)
	ReadObj(
		NETID := ADSNetId,
		PORT := 16#1000 + NodeId,
		IDXGRP := ObjectIndex,
		IDXOFFS := ObjectSubindex,
		LEN := LEN,
		DESTADDR := ADR(Data),
		READ := TRUE,
		TMOUT := t#100ms);
	iStep := 101;
101: ReadObj;
	IF NOT ReadObj.Busy THEN
		iStep := 102 ;
	END_IF
102:	IF ReadObj.Err THEN
		iStep := 0;
		ErrNo := ReadObj.ErrId;
		Multiplexor := ObjectIndex * 256; (* Shift of 8 *)
		Multiplexor := Multiplexor + ObjectSubindex;
		Err := TRUE;
	ELSE
		iStep := 0;
	END_IF;
	Done := TRUE;

ELSE
	IF Read THEN
		iStep := 1;
		Done := FALSE;
	END_IF;
END_CASE;
*)

END_FUNCTION_BLOCK

// ---- POUs/Programs/PRG_AxesEnable.TcPOU
PROGRAM PRG_AxesEnable
VAR_INPUT
	bEnable			: BOOL;	(*Enable controller*)
	bHalt			: BOOL;	(*Halt stops the axis*)
	bReset			: BOOL;	(*Resets the controller*)
END_VAR
VAR_OUTPUT
	bAxesEnabled	: BOOL;	(*All axes are enabled*)
	bFaultActive	: BOOL;	(*Fault is active on some axis*)
	wEnabledStates	: WORD;	(*Axes enable states*)
	wFaultStates	: WORD;	(*Axes fault states*)
END_VAR
VAR
	fbEnableAxis_Th1: FB_EnableAxis;
	fbEnableAxis_Th2: FB_EnableAxis;
	wMaskForAxes	: WORD := 16#03;		(*Mask for active axes in configuration*)
END_VAR

fbEnableAxis_Th1(
	bEnable:=bEnable ,
	bHalt:= bHalt,
	bReset:= bReset,
	wStatus:= GVL_AxisCtrl.AX1_diStatusWordIs,
	bEnablePos:= TRUE,
	bEnableNeg:= TRUE,
	Override:= 100,
	AxisRef := GVL_NC.Th1_AXIS,
	bDriveEnabled=> wEnabledStates.0,
	bFaultActive=> wFaultStates.0,
	wControl=>GVL_AxisCtrl.AX1_diControlWord);
	
fbEnableAxis_Th2(
	bEnable:=bEnable ,
	bHalt:= bHalt,
	bReset:= bReset,
	wStatus:= GVL_AxisCtrl.AX2_diStatusWordIs,
	bEnablePos:= TRUE,
	bEnableNeg:= TRUE,
	Override:= 100,
	AxisRef := GVL_NC.Th2_AXIS,
	bDriveEnabled=> wEnabledStates.1,
	bFaultActive=> wFaultStates.0,
	wControl=>GVL_AxisCtrl.AX2_diControlWord);


bAxesEnabled := (wEnabledStates AND wMaskForAxes) = wMaskForAxes;
bFaultActive := (wFaultStates AND wMaskForAxes) > 0;

END_PROGRAM

// ---- POUs/FB/FB_EnableAxis.TcPOU
FUNCTION_BLOCK FB_EnableAxis
VAR_INPUT
	bEnable			: BOOL;	(*Enable controller*)
	bHalt			: BOOL;	(*Halt stops the axis*)
	bReset			: BOOL;	(*Resets the controller*)
	wStatus			: WORD;	(*Status Word of the Controller*)

	bEnablePos		: BOOL;	(*Positive movement enabled*)
	bEnableNeg		: BOOL;	(*Negative movement enabled*)
	Override 		: LREAL;	(*Override for the axis*)
END_VAR
VAR_OUTPUT
	bDriveEnabled	: BOOL;	(*Controller is enabled*)
	bFaultActive	: BOOL;	(*Fault is active on controller*)
	wControl		: WORD;	(*Control word to Controller*)
END_VAR
VAR_IN_OUT
	AxisRef			: AXIS_REF;
END_VAR
VAR
	mcPower			: MC_Power;
	mcReset			: MC_Reset;
	fbEPOSControl	: FB_EPOS_Control;
	fb_Epos_SetEnabled: FB_SetEnableState;
END_VAR

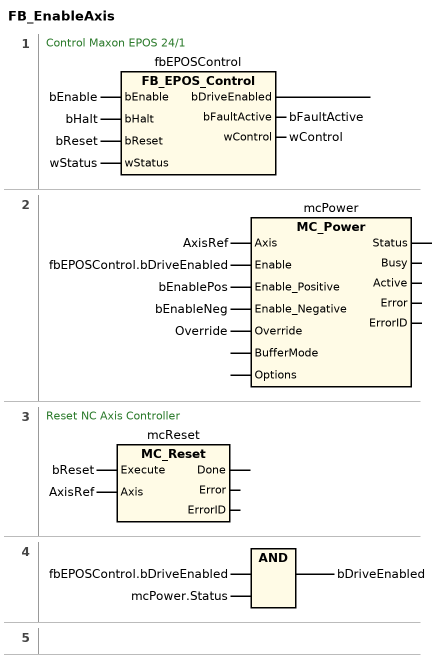
// NETWORK 1
// Control Maxon EPOS 24/1
fbEPOSControl(
    bEnable := bEnable,
    bHalt := bHalt,
    bReset := bReset,
    wStatus := wStatus,
    bFaultActive => bFaultActive,
    wControl => wControl); // FB_EPOS_Control

// NETWORK 2
mcPower(
    Axis := AxisRef,
    Enable := fbEPOSControl.bDriveEnabled,
    Enable_Positive := bEnablePos,
    Enable_Negative := bEnableNeg,
    Override := Override); // MC_Power

// NETWORK 3
// Reset NC Axis Controller
mcReset(Execute := bReset, Axis := AxisRef); // MC_Reset

// NETWORK 4
bDriveEnabled := fbEPOSControl.bDriveEnabled AND mcPower.Status;

// NETWORK 5

END_FUNCTION_BLOCK

// ---- POUs/FB/FB_EPOS_Control.TcPOU
FUNCTION_BLOCK FB_EPOS_Control
VAR_INPUT
	bEnable	: BOOL;	(*Enable controller*)
	bHalt	: BOOL;	(*Halt stops the axis*)
	bReset	: BOOL;	(*Resets the controller*)
	wStatus	: WORD;	(*Status Word of the Controller*)
END_VAR
VAR_OUTPUT
	bDriveEnabled	: BOOL;	(*Controller is enabled*)
	bFaultActive		: BOOL;	(*Fault is active on controller*)
	wControl			: WORD;	(*Control word to Controller*)
END_VAR
VAR
	iStep	: UINT;	(*Sequencer*)
	(*wControlTemp	: WORD;	(*Local temporar Control word*)*)
END_VAR


//IF wStatus.3 THEN (*Fault active*)
//	iStep := 1;
//END_IF;


//CASE iStep OF

//1:	(*Reset fault*)
//	wControl:=16#0080; (*Resets the controller from fault*)
//	IF NOT wStatus.3 THEN	(*Fault Cleared*)
//		iStep:= 2;
//	END_IF;

//2:	(*Wait for enable*)
//	IF bEnable THEN
//		iStep:= 10;
//	ELSE
//		wControl:=16#0000;	(*Disabled*)
//	END_IF;

//10:	(*Enabling procedure start*)
//	(*(Status AND Mask) = expected bit set*)
////	IF (wStatus AND 16#0017) = 16#0017 THEN
////		iStep:= 20;
////	IF wStatus.0 AND wStatus.1 AND wStatus.5 AND NOT wStatus.6 THEN
////		iStep:= 20;
//	(*(Status AND Mask) = expected bit set*)
//	IF (wStatus AND 16#0023) = 16#0023 THEN (*Switched On*)
//		iStep:= 20;
//	ELSE
//		IF wStatus.6 THEN		(*Switch on disable*)
//			iStep:= 11;
////		ELSE
////			iStep:= 20;
//		END_IF;
//	END_IF;

//11:	(*Shut down*)
//	wControl:=16#0006;
//	IF wStatus.0 THEN		(*Ready to Switch on*)
//		iStep:= 20;
//	ELSE
//		iStep:= 30;	
//	END_IF;

//20:	(*Enable operation*)
//	wControl:=16#000F;
//	IF NOT bEnable THEN		(*Disable Controller*)
//		iStep:= 2;
//	END_IF;
//30: (*Switched On*)
//	wControl := 16#0007;
//	IF wStatus.0 AND NOT wStatus.6 THEN
//		iStep:= 20;
//	END_IF

//ELSE	(*Default branch*)
//	iStep := 2;

//END_CASE;

//(*Halt control*)
//IF wStatus.2 AND NOT wStatus.1 THEN		(*Operation enabled and switched on*)
//	(*Halt active*)
//	wControl.8 :=bHalt;
//END_IF;

//(*Reset active*)
//IF bReset THEN
//	(*Resets the controller from fault*)
//	wControl:=16#0080;
//	iStep := 1;
//END_IF;

//(*Output flags*)
//bFaultActive := wStatus.3;
//bDriveEnabled := wStatus.1 AND wStatus.2;
////bDriveEnabled := TRUE;
IF NOT bEnable THEN
	iStep := 10;
END_IF

IF wStatus.3 THEN (*Fault active*)
	iStep := 1;
END_IF;

CASE iStep OF

1:	(*Reset fault*)
	wControl:=16#0080; (*Resets the controller from fault*)
	IF NOT wStatus.3 THEN	(*Fault Cleared*)
		iStep:= 10;
	END_IF;
	
10: (*State: Switch On Disable*)
	IF bEnable THEN (*Wait for enable*)
		iStep:= 20;
	ELSE
		wControl:=16#0000;	(*Switch On Disable*)	
	END_IF
	
20: (*Begin Enabling Sequence*)
	IF wStatus.6 THEN (*Switch On Disable*)	
		wControl:=16#0006;	(*Shutdown*)
	END_IF	
	IF wStatus.5 AND wStatus.0 THEN (*Ready to switch ON*) 
		wControl:=16#0007;	(*Switch On*)
	END_IF
	IF wStatus.5 AND wStatus.1 AND wStatus.0 THEN(*Switched On*)	
		iStep:= 30;
	END_IF
	
30: (*Enable operation*)
	IF NOT bEnable THEN		(*Disable Controller*)
		iStep:= 10;
	END_IF;

	IF NOT bHalt THEN
		wControl:=16#000F; 		(*Switch On & Enable Operation*)
	ELSE
		iStep:= 40;
	END_IF
		
	IF NOT wStatus.1 AND NOT wStatus.2 THEN (*Drive is not enabled*)
		iStep:= 20;
	END_IF
	
40: (*State: QuickStop Active*)
	IF bHalt THEN
		wControl := 16#0002;
	ELSE
		iStep:= 30;
	END_IF

ELSE	(*Default branch*)
	iStep := 1;

END_CASE;

(*Reset active*)
IF bReset THEN
	(*Resets the controller from fault*)
	wControl:=16#0080;
	iStep := 1;
END_IF;

(*Halt control*)
IF wStatus.2 AND NOT wStatus.1 THEN		(*Operation enabled and switched on*)
	(*Halt active*)
	wControl.8 :=bHalt;
END_IF;

(*Output flags*)
bFaultActive := wStatus.3;
bDriveEnabled := wStatus.1 AND wStatus.2;

END_FUNCTION_BLOCK

// ---- POUs/Programs/PRG_AxisControl.TcPOU
PROGRAM PRG_AxisControl
VAR
	MC_SetZero_Th1: MC_SetPosition;
	MC_SetZero_Th2: MC_SetPosition;
	MC_Jog_Th1: MC_Jog;
	MC_Jog_Th2: MC_Jog;
	MC_MoveAbsolute_Th1: MC_MoveAbsolute;
	MC_MoveAbsolute_Th2: MC_MoveAbsolute;
END_VAR

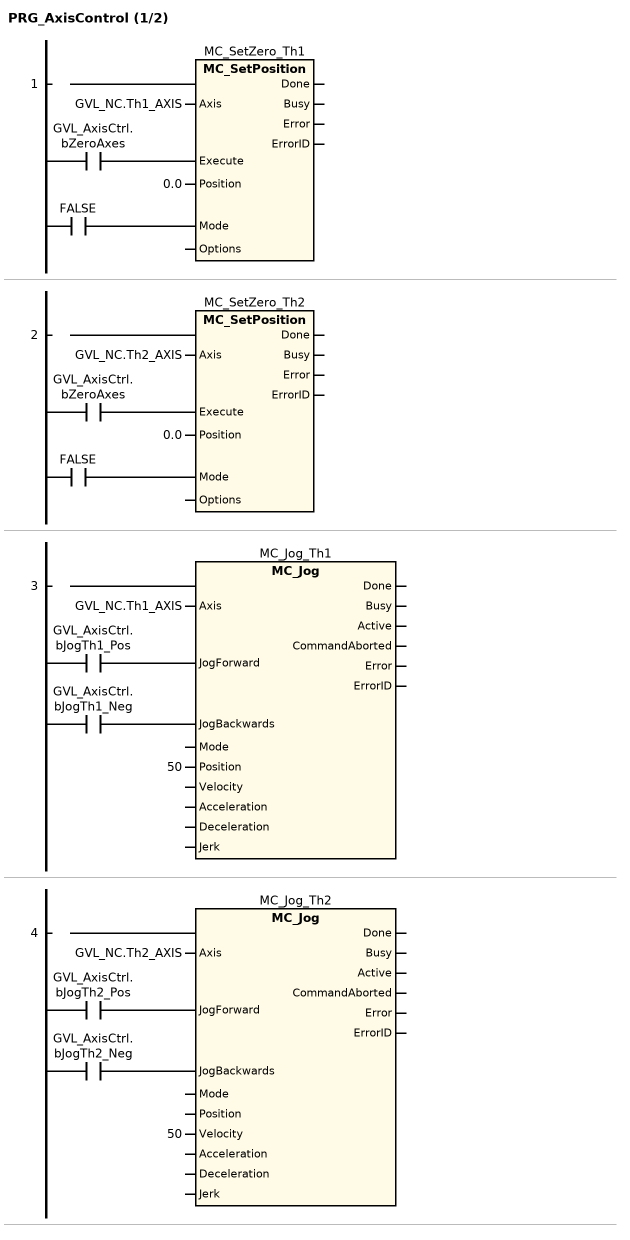
// NETWORK 1
MC_SetZero_Th1(Axis := GVL_NC.Th1_AXIS, Execute := GVL_AxisCtrl.bZeroAxes, Position := 0.0, Mode := FALSE); // MC_SetPosition

// NETWORK 2
MC_SetZero_Th2(Axis := GVL_NC.Th2_AXIS, Execute := GVL_AxisCtrl.bZeroAxes, Position := 0.0, Mode := FALSE); // MC_SetPosition

// NETWORK 3
MC_Jog_Th1(
    Axis := GVL_NC.Th1_AXIS,
    JogForward := GVL_AxisCtrl.bJogTh1_Pos,
    JogBackwards := GVL_AxisCtrl.bJogTh1_Neg,
    Position := 50); // MC_Jog

// NETWORK 4
MC_Jog_Th2(
    Axis := GVL_NC.Th2_AXIS,
    JogForward := GVL_AxisCtrl.bJogTh2_Pos,
    JogBackwards := GVL_AxisCtrl.bJogTh2_Neg,
    Velocity := 50); // MC_Jog

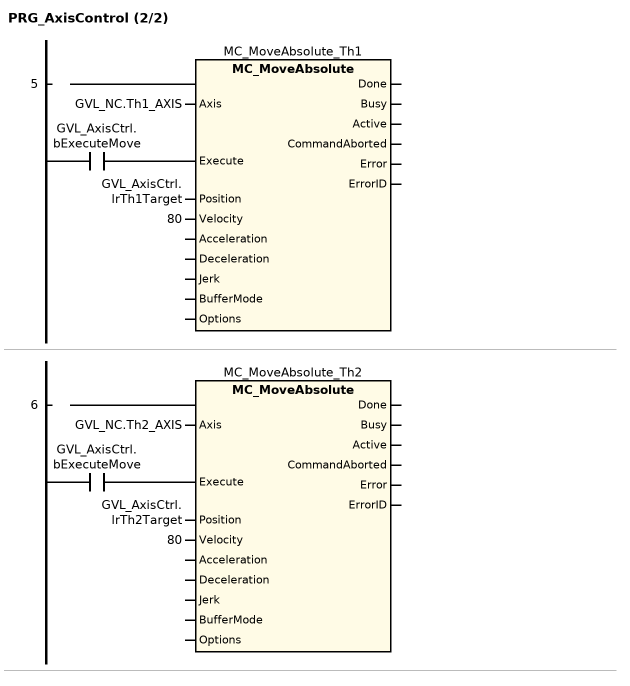
// NETWORK 5
MC_MoveAbsolute_Th1(
    Axis := GVL_NC.Th1_AXIS,
    Execute := GVL_AxisCtrl.bExecuteMove,
    Position := GVL_AxisCtrl.lrTh1Target,
    Velocity := 80); // MC_MoveAbsolute

// NETWORK 6
MC_MoveAbsolute_Th2(
    Axis := GVL_NC.Th2_AXIS,
    Execute := GVL_AxisCtrl.bExecuteMove,
    Position := GVL_AxisCtrl.lrTh2Target,
    Velocity := 80); // MC_MoveAbsolute

END_PROGRAM

// ---- POUs/Programs/PRG_updateDrives.TcPOU
PROGRAM PRG_updateDrives
VAR
END_VAR

GVL_AxisCtrl.Th1_diVeloSet_OUT := GVL_AxisCtrl.Th1_iVeloSet_IN;
GVL_AxisCtrl.Th2_diVeloSet_OUT := GVL_AxisCtrl.Th2_iVeloSet_IN;

END_PROGRAM

// ---- POUs/FB/FB_EPOSstates.TcPOU
FUNCTION_BLOCK FB_EPOSstates
VAR_INPUT
	bEnable	: BOOL;	(*Enable controller*)
	bHalt	: BOOL;	(*Halt stops the axis*)
	bReset	: BOOL;	(*Resets the controller*)
	wStatus	: WORD;	(*Status Word of the Controller*)
END_VAR
VAR_OUTPUT
	bDriveEnabled	: BOOL;	(*Controller is enabled*)
	bFaultActive		: BOOL;	(*Fault is active on controller*)
	wControl			: WORD;	(*Control word to Controller*)
END_VAR
VAR
	iStep	: UINT;	(*Sequencer*)
	(*wControlTemp	: WORD;	(*Local temporar Control word*)*)
END_VAR

IF wStatus.3 THEN (*Fault active*)
	iStep := 1;
END_IF;

CASE iStep OF

1:	(*Reset fault*)
	wControl:=16#0080; (*Resets the controller from fault*)
	IF NOT wStatus.3 THEN	(*Fault Cleared*)
		iStep:= 10;
	END_IF;
	
10: (*State: Switch On Disable*)
	IF bEnable THEN (*Wait for enable*)
		iStep:= 20;
	ELSE
		wControl:=16#0000;	(*Switch On Disable*)	
	END_IF
	
20: (*Begin Enabling Sequence*)
	IF wStatus.6 THEN (*Switch On Disable*)	
		wControl:=16#0006;	(*Shutdown*)
	END_IF	
	IF wStatus.5 AND wStatus.0 THEN (*Ready to switch ON*) 
		wControl:=16#0007;	(*Switch On*)
	END_IF
	IF wStatus.5 AND wStatus.1 AND wStatus.0 THEN(*Switched On*)	
		iStep:= 30;
	END_IF
	
30: (*Enable operation*)
	wControl:=16#000F; 		(*Switch On & Enable Operation*)
	IF NOT bEnable THEN		(*Disable Controller*)
		iStep:= 10;
	END_IF;
	
ELSE	(*Default branch*)
	iStep := 1;

END_CASE;

(*Reset active*)
IF bReset THEN
	(*Resets the controller from fault*)
	wControl:=16#0080;
	iStep := 1;
END_IF;

(*Output flags*)
bFaultActive := wStatus.3;
bDriveEnabled := wStatus.1 AND wStatus.2;

END_FUNCTION_BLOCK

// ---- POUs/FB/FB_ExtrusionSystem.TcPOU
FUNCTION_BLOCK FB_ExtrusionSystem
VAR_INPUT
	bEnable 			: BOOL;
	bReset 				: BOOL;
	bExecute			: BOOL;
	lrMMtoExtrude  		: LREAL;
	lrFeedrate   		: LREAL;
	lrHotEndTempSP		: LREAL;
	lrHotEndTemp 		: LREAL;
	
END_VAR
VAR_OUTPUT
	bDone 				: BOOL;
	sStateDesc			: STRING;
	bError				: BOOL;
	bExtruderReady		: BOOL;
	iHotEndPowerLevel 	: INT;
	bFan				: BOOL;
	bEnableHotend		: BOOL;
	
END_VAR
VAR_IN_OUT
	ExtruderAxisRef			: AXIS_REF;
END_VAR

VAR
	nState					: UDINT := 0;
	nErrorState				: UDINT;
	eErrorId				: UDINT;
	
	MC_Power_Extruder		: MC_Power;
	MC_Reset_Extruder 		: MC_Reset;
	MC_ZeroPos_Extruder		: MC_SetPosition;
	MC_Stop_Extruder 		: MC_Stop;
	MC_Move_Rel_Extruder 	: MC_MoveRelative;
	fbHotendTempController 	: FB_TempControl;
	//bEnableHotEnd: BOOL;
END_VAR

ExtruderAxisRef.ReadStatus();

MC_Power_Extruder(
	Axis:= ExtruderAxisRef, 
	Enable:= bExtruderReady, 
	Enable_Positive:= bExtruderReady, 
	Enable_Negative:= bExtruderReady, 
	Override:= , 
	BufferMode:= , 
	Options:= , 
	Status=> , 
	Busy=> , 
	Active=> , 
	Error=> bError, 
	ErrorID=> eErrorId);
	
fbHotendTempController(
		bEnableHeater:= bEnableHotEnd, 
		lrPV:= lrHotendTemp, 
		lrSP:= lrHotEndTempSP, 
		iOutput=> iHotEndPowerLevel, 
		bError=> bError, 
		eErrorId=> eErrorId,
		bEnableHotend=> bEnableHotend);
		
MC_Move_Rel_Extruder(
	Axis:= ExtruderAxisRef, 
	Execute:= GVL_AxisCtrl.bExtruder_AxisMoveHMI, 
	Distance:= GVL_AxisCtrl.lrExtruder_AxisTarget , 
	Velocity:= GVL_AxisCtrl.lrExtruder_AxisVelocity, 
	Acceleration:= , 
	Deceleration:= , 
	Jerk:= , 
	BufferMode:= , 
	Options:= , 
	Done=> GVL_AxisCtrl.bExtruder_AxisAbsMoveDone, 
	Busy=> , 
	Active=> GVL_AxisCtrl.bExtruder_AxisAbsMoveAct , 
	CommandAborted=> , 
	Error=> bError, 
	ErrorID=> eErrorId);

IF bReset THEN
	nState := 30;
END_IF

IF NOT bEnable THEN
	nState := 20;
END_IF

		
CASE nState OF
	0:	// init
		sStateDesc := 'FB INIT';
		bDone := FALSE;
		bError := FALSE;
		GVL_AxisCtrl.bExtruder_AxisAbsMove := FALSE;
		iHotEndPowerLevel := 0;
		bFan := FALSE;
		nState := 10;
		
	10:	// Init
		IF bEnable THEN 
			nState := 30;
		ELSE
			nState := 20;
		END_IF
		
	20: //Idle State
		sStateDesc := 'IDLE';
		iHotEndPowerLevel := 0;
		bEnableHotEnd := FALSE;
		bExtruderReady := FALSE;
		bFan := FALSE;
		IF bEnable THEN 
			nState := 30;
		END_IF			
		
	30:  // Reset Axis
		sStateDesc := 'RESET EXTRUDER AXIS';
		MC_Reset_Extruder(Axis:=ExtruderAxisRef, Execute:=TRUE);
		IF MC_Reset_Extruder.Done THEN
			nState := 40;
		END_IF
	
	40: // Extruder Initialised, now start heating and turn on fan
		sStateDesc := 'START HEATING';
		bEnableHotEnd := TRUE;
		bFan := TRUE;
		nState := 50;
	
	50: // Wait to reach temperature
		sStateDesc := 'WAITING TO REACH OPERATING TEMP';
		IF lrHotendTemp >= (lrHotEndTempSP*0.98) THEN
			bExtruderReady := TRUE;
			nState := 60;
		ELSE
			bExtruderReady := FALSE;
		END_IF
		
	60: // Hotened at temperature, Enable Extruder Axis
		sStateDesc := 'AT OPERATING TEMP';
		IF MC_Power_Extruder.Status THEN
			nState := 70;
		ELSE
			nState := 30;	
		END_IF
	70: // Hotened at temperature, Wait for Extrusion Command
		sStateDesc := 'WAITING FOR MOVE COMMAND';
		IF lrHotendTemp >= (lrHotEndTempSP*0.98) THEN
			bExtruderReady := TRUE;
		ELSE
			nState := 50;
		END_IF
			
	999: // Error
		sStateDesc := 'ERROR STATE';
	
	ELSE
		sStateDesc := 'INVALID STATE';
		nState := 0;
	
END_CASE

END_FUNCTION_BLOCK

// ---- POUs/Programs/PRG_ExtruderSys.TcPOU
PROGRAM PRG_ExtruderSys
VAR
	fbExtrusionSystem: FB_ExtrusionSystem;
END_VAR

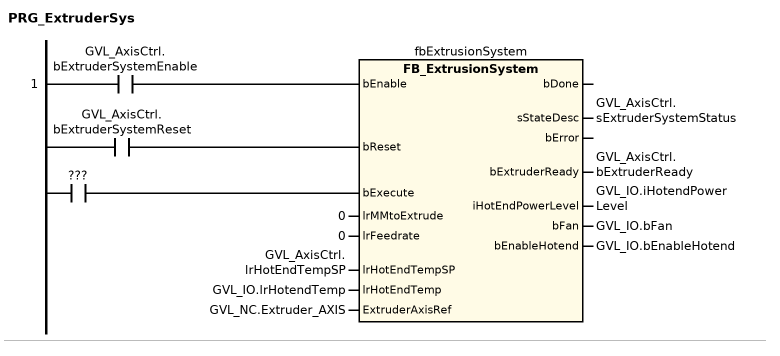
// NETWORK 1
fbExtrusionSystem(
    bEnable := GVL_AxisCtrl.bExtruderSystemEnable,
    bReset := GVL_AxisCtrl.bExtruderSystemReset,
    lrMMtoExtrude := 0,
    lrFeedrate := 0,
    lrHotEndTempSP := GVL_AxisCtrl.lrHotEndTempSP,
    lrHotEndTemp := GVL_IO.lrHotendTemp,
    ExtruderAxisRef := GVL_NC.Extruder_AXIS,
    sStateDesc => GVL_AxisCtrl.sExtruderSystemStatus,
    bExtruderReady => GVL_AxisCtrl.bExtruderReady,
    iHotEndPowerLevel => GVL_IO.iHotendPowerLevel,
    bFan => GVL_IO.bFan,
    bEnableHotend => GVL_IO.bEnableHotend); // FB_ExtrusionSystem

END_PROGRAM

// ---- GlobalTextList.TcGTLO
TEXTLIST GlobalTextList
  532 = '%10.1f'
  528 = '%s'
  56 = '+'
  866 = '-'
  636 = 'Drive Online'
  395 = 'Enable Extruder System'
  514 = 'Enable Motors'
  271 = 'Execute'
  127 = 'Extru Pos: %10.1f'
  216 = 'Extru Vel: %10.1f'
  234 = 'Extrude'
  292 = 'Extruder Filament'
  790 = 'Extruder Ready'
  950 = 'Fan On'
  201 = 'Feed Rate'
  517 = 'Feed Rate:  %10.1f'
  524 = 'Feed Rate:  %10.1f mm/s'
  430 = 'Go To Zero'
  709 = 'HE Power Level %10.1f'
  131 = 'Hot End Power Level'
  167 = 'Hotend On'
  368 = 'Hotend Setpoint'
  854 = 'MM to Extrude'
  560 = 'MM to Extrude:  %10.1f'
  187 = 'Pos: %10.1f'
  622 = 'Pos:%10.1f'
  987 = 'Power Level %10.1f'
  570 = 'Reset'
  739 = 'Setpoint: %10.1f'
  257 = 'Target'
  246 = 'Temp Set Point:  %10.1f'
  456 = 'Temp Setpoint'
  870 = 'Temp Setpoint %10.1f'
  80 = 'Temp SP:  %10.1f'
  404 = 'Temp: %10.1f'
  724 = 'Th1: %10.1f'
  737 = 'Th1:%10.1f'
  196 = 'Th2: %10.1f'
  831 = 'TH_1'
  483 = 'TH_2'
  332 = 'Vel:%10.1f'
  168 = 'Zero Axes'
END_TEXTLIST

// ---- VISUs/Visualization.TcVIS
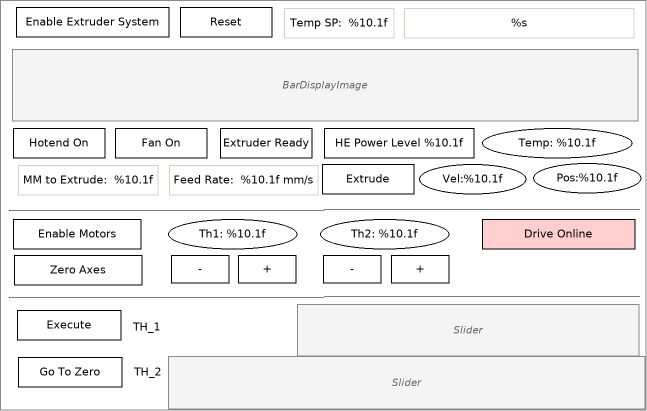
VISUALIZATION Visualization  // 647x411
    RoundedRectangle (16,7 153x30), "Enable Extruder System", colour toggle: GVL_AxisCtrl.bExtruderSystemEnable
        toggle GVL_AxisCtrl.bExtruderSystemEnable
    RoundedRectangle (13,128 92x30), "Hotend On", colour toggle: GVL_IO.bEnableHotend
    RoundedRectangle (115,128 92x30), "Fan On", colour toggle: GVL_IO.bFan
    BarDisplayImage (12,49 626x72), value: GVL_IO.lrHotendTemp, invisible if: FALSE, style: BarDisplayImage-Gray, scale format: %.1f, scale 0..300
    RoundedRectangle (180,7 92x30), "Reset"
        tap GVL_AxisCtrl.bExtruderSystemReset
        OnMouseDown: execute { GVL_AxisCtrl.bExtruderSystemEnable := FALSE; }
    Ellipse (482,128 150x30), "Temp: %10.1f", text variable: GVL_IO.lrHotendTemp
    RoundedRectangle (324,128 150x30), "HE Power Level %10.1f", text variable: GVL_IO.iHotendPowerLevel
    Textfield (284,8 110x30), "Temp SP: %10.1f", text variable: GVL_AxisCtrl.lrHotEndTempSP
        OnMouseDown: write GVL_AxisCtrl.lrHotEndTempSP via InputWithLimits, min 180, max 240
    RoundedRectangle (220,128 92x30), "Extruder Ready", colour toggle: GVL_AxisCtrl.bExtruderReady
    RoundedRectangle (322,164 92x30), "Extrude", input disabled if: NOT GVL_AxisCtrl.bExtruderReady
        tap GVL_AxisCtrl.bExtruder_AxisMoveHMI
    Textfield (404,8 230x30), "%s", text variable: GVL_AxisCtrl.sExtruderSystemStatus
    Textfield (18,165 140x30), "MM to Extrude: %10.1f", text variable: GVL_AxisCtrl.lrExtruder_AxisTarget
        OnMouseDown: write GVL_AxisCtrl.lrExtruder_AxisTarget via InputWithLimits, min 0, max 1000
    Textfield (169,165 149x30), "Feed Rate: %10.1f mm/s", text variable: GVL_AxisCtrl.lrExtruder_AxisVelocity
        OnMouseDown: write GVL_AxisCtrl.lrExtruder_AxisVelocity via InputWithLimits, min 0, max 4
    Ellipse (533,163 108x30), "Pos:%10.1f", text variable: GVL_NC.Extruder_AXIS.NcToPlc.ActPos
    Ellipse (419,164 107x30), "Vel:%10.1f", text variable: GVL_NC.Extruder_AXIS.NcToPlc.ActVelo
    Line (9,210) (639,209)
    RoundedRectangle (13,219 128x30), "Enable Motors", colour toggle: GVL_AxisCtrl.bEnableGimbal
        toggle GVL_AxisCtrl.bEnableGimbal
    RoundedRectangle (482,219 153x30), "Drive Online", colour toggle: GVL_AxisCtrl.bAllAxisEnabled
    RoundedRectangle (14,255 128x30), "Zero Axes"
        tap GVL_AxisCtrl.bZeroAxes
        OnMouseDown: execute {  }
    Ellipse (168,219 129x30), "Th1: %10.1f", text variable: GVL_NC.Th1_AXIS.NcToPlc.ActPos
    Ellipse (320,219 129x30), "Th2: %10.1f", text variable: GVL_NC.Th2_AXIS.NcToPlc.ActPos
    RoundedRectangle (171,255 58x28), "-"
        tap GVL_AxisCtrl.bJogTh1_Neg
    RoundedRectangle (391,255 58x28), "+"
        tap GVL_AxisCtrl.bJogTh2_Pos
    RoundedRectangle (238,255 58x28), "+"
        tap GVL_AxisCtrl.bJogTh1_Pos p3779583253=TRUE
    RoundedRectangle (323,255 58x28), "-"
        tap GVL_AxisCtrl.bJogTh2_Neg
    Line (9,297) (639,296)
    Slider (297,304 342x52), variable: GVL_AxisCtrl.lrTh1Target, scale -16..35
    Slider (168,356 477x53), variable: GVL_AxisCtrl.lrTh2Target, scale -160..160
    Label (122,312 50x30), "TH_1"
    RoundedRectangle (18,357 104x30), "Go To Zero"
        OnMouseDown: execute { GVL_AxisCtrl.lrTh1Target := 0; GVL_AxisCtrl.lrTh2Target := 0; GVL_AxisCtrl.bExecuteMove := TRUE; }
    Label (107,357 82x30), "TH_2"
    RoundedRectangle (17,310 104x30), "Execute"
        tap GVL_AxisCtrl.bExecuteMove
        OnMouseDown: execute {  }
END_VISUALIZATION
